SUBAPPLICATION Ventilsteuerung_Uebung_006a2 (* 2x SR&T-Flip-Flop mit IE *)
  (* Standard: 61499-2 *)
  (* Version 1.0, 2023-10-23, franz *)
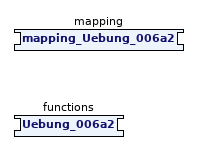
  SUBAPPS
    mapping : mapping_Uebung_006a2;
    functions : Uebung_006a2;
  END_SUBAPPS
END_SUBAPPLICATION
